// LS Electric XG5000 project: 기계실험용
// PLC NewPLC
// module base 0 slot 0: 입출력 모듈:XBM-DN32S (DC 24V 입력, 트랜지스터 출력 32점)
// module base 0 slot 1: 위치결정 모듈:XBF-PD02A (위치결정 펄스(LD)출력형, 2축)

PROGRAM NewProgram (task: 스캔 프로그램)

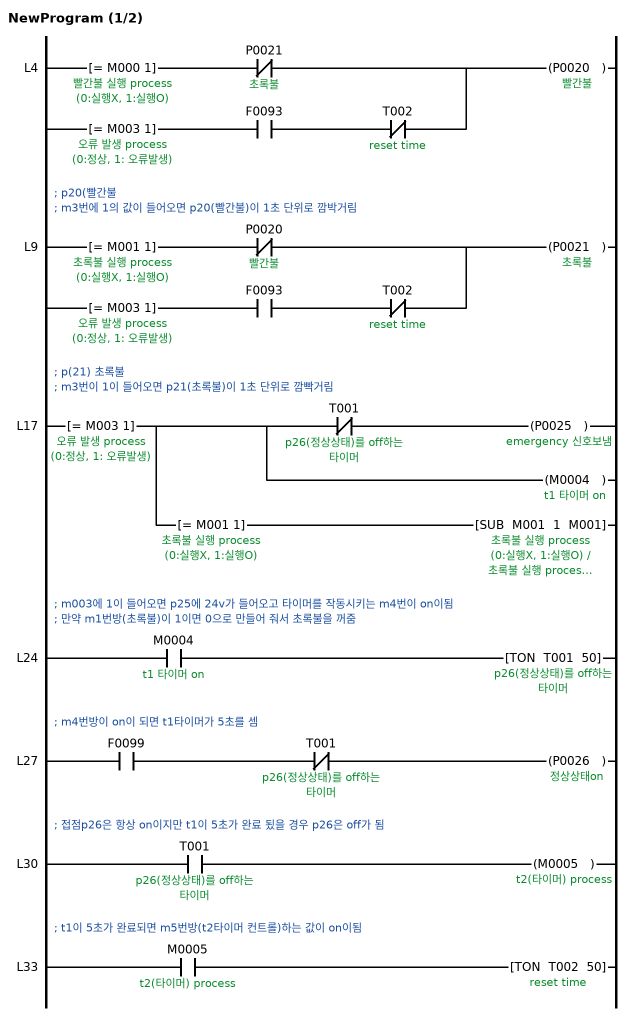
; L4
LOAD=     M000 1	// 빨간불 실행 process (0:실행X, 1:실행O)
AND NOT   P0021	// 초록불
LOAD=     M003 1	// 오류 발생 process (0:정상, 1: 오류발생)
AND       F0093
AND NOT   T002	// reset time
OR LOAD
OUT       P0020	// 빨간불
// p20(빨간불
// m3번에 1의 값이 들어오면 p20(빨간불)이 1초 단위로 깜박거림
; L9
LOAD=     M001 1	// 초록불 실행 process (0:실행X, 1:실행O)
AND NOT   P0020	// 빨간불
LOAD=     M003 1	// 오류 발생 process (0:정상, 1: 오류발생)
AND       F0093
AND NOT   T002	// reset time
OR LOAD
OUT       P0021	// 초록불
// p(21) 초록불
// m3번이 1이 들어오면 p21(초록불)이 1초 단위로 깜빡거림
; L17
LOAD=     M003 1	// 오류 발생 process (0:정상, 1: 오류발생)
MPUSH
AND NOT   T001	// p26(정상상태)를 off하는 타이머
OUT       P0025	// emergency 신호보냄
MPOP
OUT       M0004	// t1 타이머 on
AND=      M001 1	// 초록불 실행 process (0:실행X, 1:실행O)
SUB       M001 1 M001	// 초록불 실행 process (0:실행X, 1:실행O) / 초록불 실행 process (0:실행X, 1:실행O)
// m003에 1이 들어오면 p25에 24v가 들어오고 타이머를 작동시키는 m4번이 on이됨
// 만약 m1번방(초록불)이 1이면 0으로 만들어 줘서 초록불을 꺼줌
; L24
LOAD      M0004	// t1 타이머 on
TON       T001 50	// p26(정상상태)를 off하는 타이머
// m4번방이 on이 되면 t1타이머가 5초를 셈
; L27
LOAD      F0099
AND NOT   T001	// p26(정상상태)를 off하는 타이머
OUT       P0026	// 정상상태on
// 접점p26은 항상 on이지만 t1이 5초가 완료 됬을 경우 p26은 off가 됨
; L30
LOAD      T001	// p26(정상상태)를 off하는 타이머
OUT       M0005	// t2(타이머) process
// t1이 5초가 완료되면 m5번방(t2타이머 컨트롤)하는 값이 on이됨
; L33
LOAD      M0005	// t2(타이머) process
TON       T002 50	// reset time

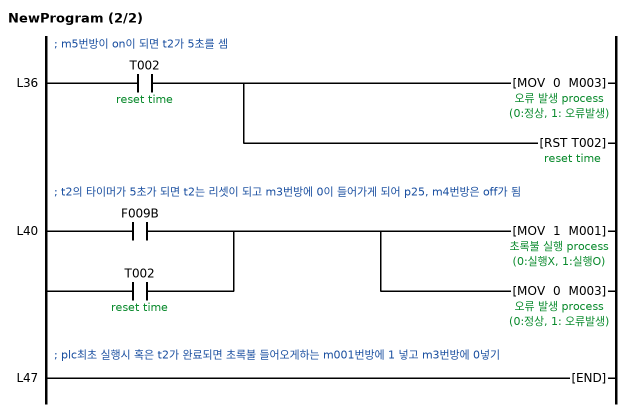
// m5번방이 on이 되면 t2가 5초를 셈
; L36
LOAD      T002	// reset time
MOV       0 M003	// 오류 발생 process (0:정상, 1: 오류발생)
RST       T002	// reset time
// t2의 타이머가 5초가 되면 t2는 리셋이 되고 m3번방에 0이 들어가게 되어 p25, m4번방은 off가 됨
; L40
LOAD      F009B
OR        T002	// reset time
MOV       1 M001	// 초록불 실행 process (0:실행X, 1:실행O)
MOV       0 M003	// 오류 발생 process (0:정상, 1: 오류발생)
// plc최초 실행시 혹은 t2가 완료되면 초록불 들어오게하는 m001번방에 1 넣고 m3번방에 0넣기
; L47
END